KUKA KRL program: TipDress_1.src, TipDress_1.dat

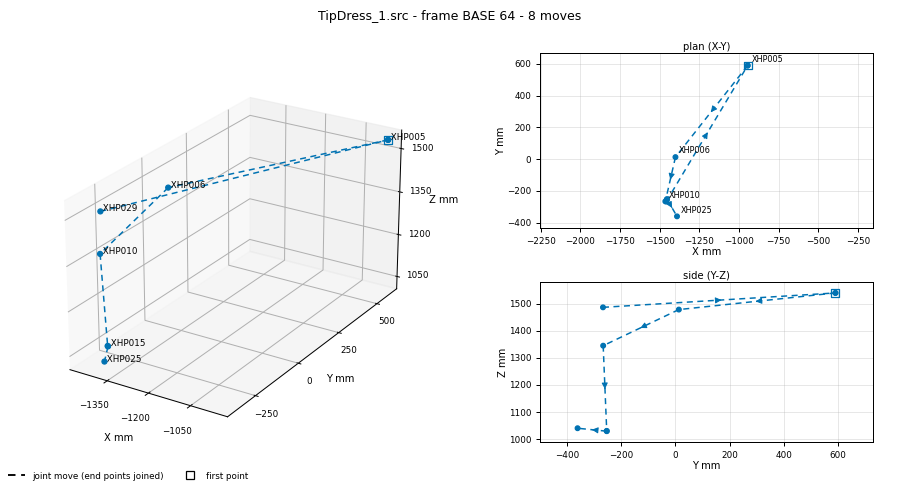
[picture p0: tool path of TipDress_1.src in frame BASE 64, 8 of 14 moves have a stored position in this frame; points joined in program order, loops and branches not executed]
--- TipDress_1.src ---
&ACCESS RVP
&REL 14
&COMMENT Kappenfraesen
&PARAM DISKPATH = KRC:\R1\Service
DEF TipDress_1( )
;FOLD INI;%{PE}
  ;FOLD BASISTECH INI
    GLOBAL INTERRUPT DECL 3 WHEN $STOPMESS==TRUE DO IR_STOPM ( )
    INTERRUPT ON 3
    BAS (#INITMOV,0 )
  ;ENDFOLD (BASISTECH INI)
  ;FOLD USER INI
    ;Make your modifications here
  ;ENDFOLD (USER INI)
;ENDFOLD (INI)
;FOLD ; Anlagenbezeichn: HC51_B    Stations-Nr: 040RB_100;%{PE}
;FOLD Parameters ;%{h}
;Params IlfProvider=kukaroboter.basistech.inlineforms.comments.comment; Kuka.Content=Anlagenbezeichn: HC51_B    Stations-Nr: 040RB_100
;ENDFOLD
;ENDFOLD
;FOLD ; Stand / Version: V1.0;%{PE}
;FOLD Parameters ;%{h}
;Params IlfProvider=kukaroboter.basistech.inlineforms.comments.comment; Kuka.Content=Stand / Version: V1.0
;ENDFOLD
;ENDFOLD
;FOLD ; Name Bearbeiter: EBZ-AE;%{PE}
;FOLD Parameters ;%{h}
;Params IlfProvider=kukaroboter.basistech.inlineforms.comments.comment; Kuka.Content=Name Bearbeiter: EBZ-AE
;ENDFOLD
;ENDFOLD
;FOLD ; Translator Version:29.01.2024 - Version 15.08;%{PE}
;FOLD Parameters ;%{h}
;Params IlfProvider=kukaroboter.basistech.inlineforms.comments.comment; Kuka.Content=Translator Version:29.01.2024 - Version 15.08
;ENDFOLD
;ENDFOLD

;Collision detection - Global/HOME/Guebergabe
;FOLD COLLDETECT UseDataSet DataSet[30];%{PE}%R 8.5.19,%MKUKATPBASIS,%CTQ_MON,%VTQ_CDSET,%P 2:TQ_CDSET, 4:30
USE_CD_PARAMS( 30)
;ENDFOLD

WAIT FOR FALSE ;STATUS
;FOLD ; 23.08.24 10:54 NAME: BS CHANGES: Pogram teached and checked T1 ;%{PE}
;FOLD Parameters ;%{h}
;Params IlfProvider=kukaroboter.basistech.inlineforms.comments.datetimecomment; Kuka.DateTime=23.08.24 10:54; Kuka.Name=BS; Kuka.Content=Pogram teached and checked T1
;ENDFOLD
;ENDFOLD
;COLLISIONS NOT CHECKED

WAIT FOR DSG_nearE6Axis (XHOME)
;FOLD PTP HOME Vel=100 % DEFAULT;%{PE}
;FOLD Parameters ;%{h}
;Params IlfProvider=kukaroboter.basistech.inlineforms.movement.old; Kuka.IsGlobalPoint=False; Kuka.PointName=HOME; Kuka.BlendingEnabled=False; Kuka.MoveDataPtpName=DEFAULT; Kuka.VelocityPtp=100; Kuka.CurrentCDSetIndex=0; Kuka.MovementParameterFieldEnabled=True; IlfCommand=PTP
;ENDFOLD
$BWDSTART = FALSE
PDAT_ACT = PDEFAULT
FDAT_ACT = FHOME
BAS(#PTP_PARAMS, 100.0)
SET_CD_PARAMS (0)
PTP XHOME
;ENDFOLD

;Collision detection - TipDress/Special Functions
;FOLD COLLDETECT UseDataSet DataSet[29];%{PE}%R 8.5.19,%MKUKATPBASIS,%CTQ_MON,%VTQ_CDSET,%P 2:TQ_CDSET, 4:29
USE_CD_PARAMS( 29)
;ENDFOLD

;// -- Kuehlwasser ein  --
;FOLD Switch Cooling Water ON
Water_ON(intGunNo)
;ENDFOLD

;FOLD DSG_.Init --> Daimler_ServoGun Init ;%{PE}
 Dsg_Process(#DSG_Init )  ;	--> Basic Setup
;ENDFOLD

;FOLD DSG_Gun_.Mode : 1 , CMD: Activate ;%{PE}%
 Wait For Dsg_Gun_Change( 1, #FastActivate)
;ENDFOLD

;FOLD PTP HP005 CONT Vel=100 % PDAT2 Tool[1]:SWZ_01_X Base[64]:Zero;%{PE}
;FOLD Parameters ;%{h}
;Params IlfProvider=kukaroboter.basistech.inlineforms.movement.old; Kuka.IsGlobalPoint=False; Kuka.PointName=HP005; Kuka.BlendingEnabled=True; Kuka.MoveDataPtpName=PDAT2; Kuka.VelocityPtp=100; Kuka.CurrentCDSetIndex=0; Kuka.MovementParameterFieldEnabled=True; IlfCommand=PTP
;ENDFOLD
$BWDSTART = FALSE
PDAT_ACT = PPDAT2
FDAT_ACT = FHP005
BAS(#PTP_PARAMS, 100.0)
SET_CD_PARAMS (0)
PTP XHP005 C_Dis
;ENDFOLD
;FOLD PTP HP006 CONT Vel=100 % PDAT5 Tool[1]:SWZ_01_X Base[64]:Zero ;%{PE}
;FOLD Parameters ;%{h}
;Params IlfProvider=kukaroboter.basistech.inlineforms.movement.old; Kuka.IsGlobalPoint=False; Kuka.PointName=HP006; Kuka.BlendingEnabled=True; Kuka.MoveDataPtpName=PDAT5; Kuka.VelocityPtp=100; Kuka.CurrentCDSetIndex=0; Kuka.MovementParameterFieldEnabled=True; IlfCommand=PTP
;ENDFOLD
$BWDSTART = FALSE
PDAT_ACT = PPDAT5
FDAT_ACT = FHP006
BAS(#PTP_PARAMS, 100.0)
SET_CD_PARAMS (0)
PTP XHP006 C_Dis
;ENDFOLD
;FOLD PTP HP010 CONT Vel=100 % PDAT3 Tool[1]:SWZ_01_X Base[64]:Zero;%{PE}
;FOLD Parameters ;%{h}
;Params IlfProvider=kukaroboter.basistech.inlineforms.movement.old; Kuka.IsGlobalPoint=False; Kuka.PointName=HP010; Kuka.BlendingEnabled=True; Kuka.MoveDataPtpName=PDAT3; Kuka.VelocityPtp=100; Kuka.CurrentCDSetIndex=0; Kuka.MovementParameterFieldEnabled=True; IlfCommand=PTP
;ENDFOLD
$BWDSTART = FALSE
PDAT_ACT = PPDAT3
FDAT_ACT = FHP010
BAS(#PTP_PARAMS, 100.0)
SET_CD_PARAMS (0)
PTP XHP010 C_Dis
;ENDFOLD

REPEAT

;FOLD PTP HP015 Vel=100 % PDAT4 Tool[1]:SWZ_01_X Base[64]:Zero;%{PE}
;FOLD Parameters ;%{h}
;Params IlfProvider=kukaroboter.basistech.inlineforms.movement.old; Kuka.IsGlobalPoint=False; Kuka.PointName=HP015; Kuka.BlendingEnabled=False; Kuka.MoveDataPtpName=PDAT4; Kuka.VelocityPtp=100; Kuka.CurrentCDSetIndex=0; Kuka.MovementParameterFieldEnabled=True; IlfCommand=PTP
;ENDFOLD
$BWDSTART = FALSE
PDAT_ACT = PPDAT4
FDAT_ACT = FHP015
BAS(#PTP_PARAMS, 100.0)
SET_CD_PARAMS (0)
PTP XHP015
;ENDFOLD

;FOLD DSG_Dress._LIN DressGun_1, Vel= 0.5 m/s,  CPDAT5, ServoGun=1, Tool.[1], SWZ_01_X, Base.[64], Zero, EXT.TCP=FALSE, ;%{PE}
$BWDSTART=FALSE
LDAT_ACT=LCPDAT5
FDAT_ACT=DSG_FDAT_T(SDressGun_1)
DSG_ACT=DSG_PAR(SDressGun_1)
BAS(#CP_PARAMS,0.5)
DSG_SPOT_POINT=DSG_POS(xDressGun_1,"L" ,oDressGun_1)
LIN DSG_SPOT_POINT
DSG_Swivel_To_WorkPos ( )
DSG_Process(#Dsg_Dress  )
DSG_Swivel_To_HOMEPos ( )
LIN DSG_SPOT_POINT
DSG_Process(#DSG_POST )
;ENDFOLD

;FOLD LIN HP020 Vel=0.2 m/s CPDAT6 Tool[1]:SWZ_01_X Base[64]:Zero ;%{PE}
;FOLD Parameters ;%{h}
;Params IlfProvider=kukaroboter.basistech.inlineforms.movement.old; Kuka.IsGlobalPoint=False; Kuka.PointName=HP020; Kuka.BlendingEnabled=False; Kuka.MoveDataName=CPDAT6; Kuka.VelocityPath=0.2; Kuka.CurrentCDSetIndex=0; Kuka.MovementParameterFieldEnabled=True; IlfCommand=LIN
;ENDFOLD
$BWDSTART = FALSE
LDAT_ACT = LCPDAT6
FDAT_ACT = FHP020
BAS(#CP_PARAMS, 0.2)
SET_CD_PARAMS (0)
LIN XHP020
;ENDFOLD

 ;// -- Bewegungen aus dem Fraeser --
;FOLD PTP HP025 CONT Vel=100 % PDAT7 Tool[1]:SWZ_01_X Base[64]:Zero;%{PE}
;FOLD Parameters ;%{h}
;Params IlfProvider=kukaroboter.basistech.inlineforms.movement.old; Kuka.IsGlobalPoint=False; Kuka.PointName=HP025; Kuka.BlendingEnabled=True; Kuka.MoveDataPtpName=PDAT7; Kuka.VelocityPtp=100; Kuka.CurrentCDSetIndex=0; Kuka.MovementParameterFieldEnabled=True; IlfCommand=PTP
;ENDFOLD
$BWDSTART = FALSE
PDAT_ACT = PPDAT7
FDAT_ACT = FHP025
BAS(#PTP_PARAMS, 100.0)
SET_CD_PARAMS (0)
PTP XHP025 C_Dis
;ENDFOLD

;FOLD DSG_Ini_Tip.Gun : 1, Set Mode: Non , With Measure: Yes;%{PE}%
 Dsg_Ini_Tip( 1, #NON, True)
 ;ENDFOLD

;FOLD DSG_Ref._Weld  WeldGun_1, Vel= 100  %,  PDAT8, ServoGun= 1  , Tool[1], SWZ_01_X, Base[64], Zero, EXT.TCP= FALSE,  ;%{PE}
$BWDSTART=FALSE
PDAT_ACT=PPDAT8
FDAT_ACT=DSG_FDAT_T(SWeldGun_1)
DSG_ACT=DSG_PAR(SWeldGun_1)
BAS(#PTP_PARAMS,100)
ACT_CMD=#Dsg_RefWeld
DSG_SPOT_POINT=xWeldGun_1
PTP DSG_SPOT_POINT
DSG_Process(#Dsg_RefWeld  )
PTP DSG_SPOT_POINT
;ENDFOLD

;// -- Pruefen Fraesung OK

UNTIL DSG_Check_TipDress_OK ( Dsg_act_Gun)

;// -- Bewegungen zur HOME position --

;FOLD PTP HP029 CONT Vel=100 % PDAT6 Tool[1]:SWZ_01_X Base[64]:Zero ;%{PE}
;FOLD Parameters ;%{h}
;Params IlfProvider=kukaroboter.basistech.inlineforms.movement.old; Kuka.IsGlobalPoint=False; Kuka.PointName=HP029; Kuka.BlendingEnabled=True; Kuka.MoveDataPtpName=PDAT6; Kuka.VelocityPtp=100; Kuka.CurrentCDSetIndex=0; Kuka.MovementParameterFieldEnabled=True; IlfCommand=PTP
;ENDFOLD
$BWDSTART = FALSE
PDAT_ACT = PPDAT6
FDAT_ACT = FHP029
BAS(#PTP_PARAMS, 100.0)
SET_CD_PARAMS (0)
PTP XHP029 C_Dis
;ENDFOLD
;FOLD PTP HP030 CONT Vel=100 % PDAT9 Tool[1]:SWZ_01_X Base[64]:Zero;%{PE}
;FOLD Parameters ;%{h}
;Params IlfProvider=kukaroboter.basistech.inlineforms.movement.old; Kuka.IsGlobalPoint=False; Kuka.PointName=HP030; Kuka.BlendingEnabled=True; Kuka.MoveDataPtpName=PDAT9; Kuka.VelocityPtp=100; Kuka.CurrentCDSetIndex=0; Kuka.MovementParameterFieldEnabled=True; IlfCommand=PTP
;ENDFOLD
$BWDSTART = FALSE
PDAT_ACT = PPDAT9
FDAT_ACT = FHP030
BAS(#PTP_PARAMS, 100.0)
SET_CD_PARAMS (0)
PTP XHP030 C_Dis
;ENDFOLD

;Collision detection - Global/HOME/Guebergabe
;FOLD COLLDETECT UseDataSet DataSet[30];%{PE}%R 8.5.19,%MKUKATPBASIS,%CTQ_MON,%VTQ_CDSET,%P 2:TQ_CDSET, 4:30
USE_CD_PARAMS( 30)

;ENDFOLD

;FOLD PTP HOME Vel=100 % DEFAULT;%{PE}
;FOLD Parameters ;%{h}
;Params IlfProvider=kukaroboter.basistech.inlineforms.movement.old; Kuka.IsGlobalPoint=False; Kuka.PointName=HOME; Kuka.BlendingEnabled=False; Kuka.MoveDataPtpName=DEFAULT; Kuka.VelocityPtp=100; Kuka.CurrentCDSetIndex=0; Kuka.MovementParameterFieldEnabled=True; IlfCommand=PTP
;ENDFOLD
$BWDSTART = FALSE
PDAT_ACT = PDEFAULT
FDAT_ACT = FHOME
BAS(#PTP_PARAMS, 100.0)
SET_CD_PARAMS (0)
PTP XHOME
;ENDFOLD

 ;Collision detection - Off
 ;FOLD COLLDETECT Off ;%{PE}
 ;FOLD Parameters ;%{h}
 ;Params IlfProvider=kukaroboter.basistech.inlineforms.colldetect.off; CollDetect.Command=Off
 ;ENDFOLD
 USE_CD_PARAMS(0)
 ;ENDFOLD
END

--- TipDress_1.dat ---
&ACCESS  RVP
&COMMENT Kappenfraesen
&PARAM DISKPATH = KRC:\R1\Service
&REL 2
DEFDAT  TIPDRESS_1
;FOLD EXTERNAL DECLARATIONS;%{PE}%MKUKATPBASIS,%CEXT,%VCOMMON,%P
;FOLD BASISTECH EXT;%{PE}%MKUKATPBASIS,%CEXT,%VEXT,%P
EXT  BAS (BAS_COMMAND  :IN,REAL  :IN )
DECL INT SUCCESS
;ENDFOLD (BASISTECH EXT)
;FOLD USER EXT;%{E}%MKUKATPUSER,%CEXT,%VEXT,%P
;Make your modifications here
;ENDFOLD (USER EXT)
;FOLD COLLISION
EXT  COLLSTOP (INT  :IN,INT  :IN )
;ENDFOLD  (Collision)
;ENDFOLD (EXTERNAL DECLERATIONS)
;//-- Default Dai_ILF Structure SpotWeld --
DECL DSG_Simple_para_T DSG_Simple_para_TDefault={GunNo 1,EQ_Para 3} ;// iW6
;//-- Default Dai_ILF Structure SpotWeld --

DECL DSG_OFFSET_T oWeldGun_1={M #Base_,X 0.0,Y 0.0,Z 0.0}
DECL DSG_TIMER_TYP_T DSGWeldGun_1={PointName[] "PointName",Weld_Force 1.00000,Part_Thickness 5.00000,Weld_Time -1.00000,Gun_Deflect 0.0,Turn_Ang 0.0,Turn_TiAct 0,Turn_TiPre 0,EQ_Sens 0.0}
DECL DSG_FDAT_T SWeldGun_1={EQ_Sens 0.0,GUN_ID 1,Par_T 0,POINT_ID 99999999,Par_R 1,Par_S 0,Par_Q 1,CONT FALSE,Tool_No 1,Base_No 64,Ipo_Frame #BASE,PoINT2[] "/ ",Tq_State FALSE}
DECL DSG_Simple_para_T s_WeldGun_1={GunNo 1,EQ_Para 3,intPar1 1,intPar2 1,intPar3 1}
DECL T_MoveType miWeldGun_1={MoveType #PTP_Move,ContType #C_NotActive,charProgID[] "99999999",OnOpen 2,OnTouchUp 1,OnAccept 2}
; BASIS_SUGG_T declarations
DECL BASIS_SUGG_T LAST_BASIS={POINT1[] "P0                      ",POINT2[] "P0                      ",CP_PARAMS[] "CPDAT0                  ",PTP_PARAMS[] "PDAT0                   ",CONT[] "                        ",CP_VEL[] "2.0                     ",PTP_VEL[] "100                     ",SYNC_PARAMS[] "SYNCDAT                 ",SPL_NAME[] "S0                      ",A_PARAMS[] "ADAT0                   "}
; E6POS declarations
DECL E6POS XHP005={X -945.200500,Y 589.862366,Z 1539.13477,A -73.0697403,B 107.054741,C -74.1934280,S 18,T 11,E1 -250.000,E2 0.0,E3 0.0,E4 0.0,E5 0.0,E6 0.0}
DECL E6POS XHP010={X -1464.02039,Y -266.395386,Z 1344.69556,A -45.0001450,B 97.0000076,C -89.9999390,S 18,T 11,E1 -250.000,E2 0.0,E3 0.0,E4 0.0,E5 0.0,E6 0.0}
DECL E6POS XHP015={X -1454.54797,Y -253.321579,Z 1030.65454,A 134.990082,B 79.9983597,C 89.9896393,S 18,T 11,E1 -100.000,E2 0.0,E3 0.0,E4 0.0,E5 0.0,E6 0.0}
DECL E6POS XDressGun_1={X -1418.11511,Y -218.106934,Z 1029.30432,A 134.993164,B 80.0014725,C 89.9929733,S 18,T 11,E1 -99.9954071,E2 0.0,E3 0.0,E4 0.0,E5 0.0,E6 0.0}
DECL E6POS XHP020={X -1453.29126,Y -253.193207,Z 1029.42810,A 134.984039,B 79.9987335,C 89.9835892,S 18,T 11,E1 -99.9954071,E2 0.0,E3 0.0,E4 0.0,E5 0.0,E6 0.0}
DECL E6POS XHP025={X -1390.47131,Y -360.830,Z 1040.38074,A 148.771,B 87.7706223,C 111.597961,S 18,T 11,E1 -99.9954071,E2 0.0,E3 0.0,E4 0.0,E5 0.0,E6 0.0}
DECL E6POS XWeldGun_1={X -1391.69788,Y -361.756805,Z 1040.39502,A 148.760147,B 87.7706604,C 111.587135,S 18,T 11,E1 -99.9954071,E2 0.0,E3 0.0,E4 0.0,E5 0.0,E6 0.0}
DECL E6POS XHP030={X -945.201782,Y 589.861328,Z 1539.13513,A -73.0695572,B 107.054832,C -74.1933517,S 18,T 11,E1 -250.000,E2 0.0,E3 0.0,E4 0.0,E5 0.0,E6 0.0}
; FDAT declarations
DECL FDAT FHOME={TOOL_NO 1,BASE_NO 64,IPO_FRAME #BASE,POINT2[] " "}
DECL FDAT FHP005={TOOL_NO 1,BASE_NO 64,IPO_FRAME #BASE,POINT2[] " "}
DECL FDAT FHP010={TOOL_NO 1,BASE_NO 64,IPO_FRAME #BASE,POINT2[] " "}
DECL FDAT FHP015={TOOL_NO 1,BASE_NO 64,IPO_FRAME #BASE,POINT2[] " "}
DECL FDAT FDressGun_1={TOOL_NO 1,BASE_NO 64,IPO_FRAME #BASE,POINT2[] " "}
DECL FDAT FHP020={TOOL_NO 1,BASE_NO 64,IPO_FRAME #BASE,POINT2[] " "}
DECL FDAT FHP025={TOOL_NO 1,BASE_NO 64,IPO_FRAME #BASE,POINT2[] " "}
DECL FDAT FWeldGun_1={TOOL_NO 1,BASE_NO 64,IPO_FRAME #BASE}
DECL FDAT FHP030={TOOL_NO 1,BASE_NO 64,IPO_FRAME #BASE,POINT2[] " "}
; FRAME declarations
DECL FRAME ofWeldGun_1={X 0.0,Y 0.0,Z 0.0,A 0.0,B 0.0,C 0.0}
; LDAT declarations
DECL LDAT LCPDAT5={VEL 0.200000,ACC 100.000,APO_DIST 0.0,APO_FAC 50.0000,AXIS_VEL 100.000,AXIS_ACC 100.000,ORI_TYP #VAR,CIRC_TYP #BASE,JERK_FAC 50.0000,GEAR_JERK 50.0000,EXAX_IGN 0}
DECL LDAT LCPDAT6={VEL 0.200000,ACC 100.000,APO_DIST 0.0,APO_FAC 50.0000,AXIS_VEL 100.000,AXIS_ACC 100.000,ORI_TYP #VAR,CIRC_TYP #BASE,JERK_FAC 50.0000,GEAR_JERK 50.0000,EXAX_IGN 0}
; MODULEPARAM_T declarations
DECL MODULEPARAM_T LAST_TP_PARAMS={PARAMS[] "Kuka.VelocityPtp=100; Kuka.BlendingEnabled=True; Kuka.CurrentCDSetIndex=0; Dai.IlfConfig=DaiWeldIlfConfig.xml; Dai.IlfTech=DSG_Weld; Kuka.PointName=HP029; Kuka.FrameData.base_no=64; Kuka.FrameData.tool_no=1; Kuka.FrameData.ipo_frame=#BASE; Kuka.FrameData.point2=; Kuka.isglobalpoint=False; Kuka.MoveDataPtpName=PDAT6; Kuka.MovementDataPdat.apo_mode=#CDIS; Kuka.MovementDataPdat.apo_dist=0; Kuka.MovementData.vel=100; Kuka.MovementData.acc=100; Kuka.MovementData.gear_jerk=100; Kuka.MovementData.exax_ign=0; DSG_REF.DSG_FRAMELIST=WeldGun_1; DSG_REF.DSG_P_VEL=100; DSG_REF.DSG_PL_PDAT=PDAT8; DSG_REF.DSG_GUN=1; DSG_REF.DSG_PTOOL_ID=Tool[1]; DSG_REF.DSG_PTOOLNAME=SWZ_01_X; DSG_REF.DSG_PBASE_ID=Base[64]; DSG_REF.DSG_PBASENAME=Zero; DSG_REF.IPO_FRAME=#BASE; DSG_REF.DSG_TORQACTIVE=; Kuka.APXEnabled=False; Kuka.Name=BS; Kuka.Content=Pogram teached and checked T1"}
; PDAT declarations
DECL PDAT PPDAT1={VEL 100.000,ACC 100.000,APO_DIST 0.0,APO_MODE #CDIS,GEAR_JERK 50.0000,EXAX_IGN 0}
DECL PDAT PPDAT2={VEL 100.000,ACC 100.000,APO_DIST 1000.00,APO_MODE #CDIS,GEAR_JERK 50.0000,EXAX_IGN 0}
DECL PDAT PPDAT3={VEL 100.000,ACC 100.000,APO_DIST 1000.00,APO_MODE #CDIS,GEAR_JERK 50.0000,EXAX_IGN 0}
DECL PDAT PPDAT4={VEL 100.000,ACC 100.000,APO_DIST 0.0,APO_MODE #CDIS,GEAR_JERK 50.0000,EXAX_IGN 0}
DECL PDAT PPDAT7={VEL 100.000,ACC 100.000,APO_DIST 1000.00,APO_MODE #CDIS,GEAR_JERK 50.0000,EXAX_IGN 0}
DECL PDAT PPDAT8={VEL 100.000,ACC 100.000,APO_DIST 1.00000,APO_MODE #CDIS,GEAR_JERK 50.0000,EXAX_IGN 0}
DECL PDAT PPDAT9={VEL 100.000,ACC 100.000,APO_DIST 1000.00,APO_MODE #CDIS,GEAR_JERK 50.0000,EXAX_IGN 0}
DECL PDAT PPDAT10={VEL 100.000,ACC 100.000,APO_DIST 0.0,APO_MODE #CDIS,GEAR_JERK 50.0000,EXAX_IGN 0}
DECL DSG_OFFSET_T ODressGun_1={M #Base_,X 0.0,Y 0.0,Z 0.0}
DECL DSG_FDAT_T SDressGun_1={EQ_Sens 0.0,GUN_ID 1,Par_T 0,POINT_ID 99999999,Par_R 1,Par_S 0,Par_Q 1,CONT FALSE,Tool_No 1,Base_No 64,Ipo_Frame #BASE,PoINT2[] "/ ",Tq_State FALSE}

DECL E6POS XHP006={X -1400.33386,Y 12.6068163,Z 1477.82239,A 136.998672,B 78.1689301,C 102.228706,S 18,T 11,E1 -250.000,E2 0.0,E3 0.0,E4 0.0,E5 0.0,E6 0.0}
DECL FDAT FHP006={TOOL_NO 1,BASE_NO 64,IPO_FRAME #BASE,POINT2[] " "}
DECL PDAT PPDAT5={VEL 100.000,ACC 100.000,APO_DIST 1000.00,APO_MODE #CDIS,GEAR_JERK 50.0000,EXAX_IGN 0}
DECL PDAT P_TEMP={VEL 100.000,ACC 100.000,APO_DIST 1.00000,APO_MODE #CPTP}
DECL LDAT L_TEMP={VEL 2.00000,ACC 100.000,APO_DIST 1.00000,APO_FAC 50.0000,ORI_TYP #VAR}
DECL FDAT IPO_TEMP={IPO_FRAME #BASE}
DECL E6POS XHP029={X -1458.00745,Y -267.076233,Z 1486.06445,A 153.972351,B 77.1255493,C 109.220963,S 18,T 11,E1 -250.000,E2 0.0,E3 0.0,E4 0.0,E5 0.0,E6 0.0}
DECL FDAT FHP029={TOOL_NO 1,BASE_NO 64,IPO_FRAME #BASE,POINT2[] " "}
DECL PDAT PPDAT6={VEL 100.000,ACC 100.000,APO_DIST 0.0,APO_MODE #CDIS,GEAR_JERK 100.000,EXAX_IGN 0}
ENDDAT
